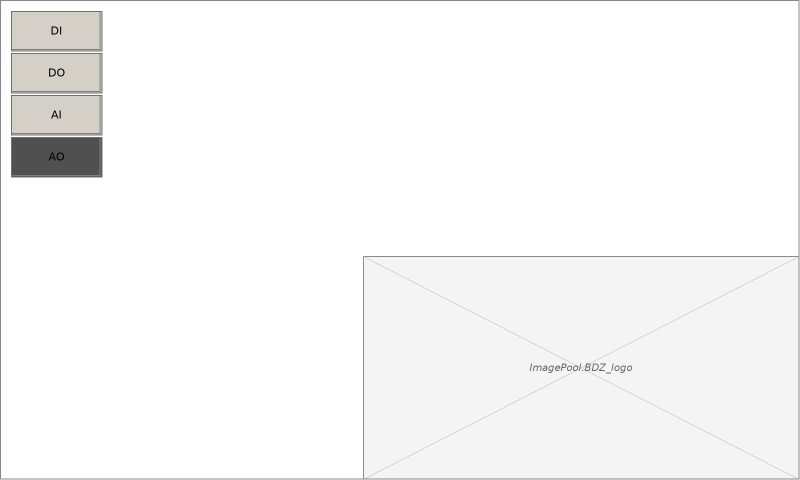
VISUALIZATION Visualization  // 800x480
    Image (363,256 436x223), image: ImagePool.BDZ_logo
    Button (11,11 91x40), "DI"
        OnMouseUp: change screen: Digital_Inputs
    Button (11,53 91x40), "DO"
        OnMouseDown: change screen: Digital_Outputs
        OnMouseUp: change screen: Digital_Outputs
    Button (11,95 91x40), "AI"
        OnMouseUp: change screen: Analog_Inputs
    Button (11,137 91x40), "AO"
        OnMouseUp: change screen: Analog_Outputs
END_VISUALIZATION

(* stored: Version 1.1.0.1, ProductVersion 3.1.4024.4
   Visu Visualization: Id {6d193410-feec-4289-ab3a-547d8676ecab} *)
